FUNCTION_BLOCK FB_HE_SATT_FilterHolderTestDouble IMPLEMENTS I_HE_SATT_FilterHolder
VAR
    nNumberOfSlots : INT;
    aiFilter : ARRAY[1..PL_HE_SATT_Parameters.nMaxNumFiltersPerHolder] Of I_HE_SATT_Filter;
END_VAR


METHOD PUBLIC GetFilter : I_HE_SATT_Filter
VAR_INPUT
	nFilterNumber	: INT;
END_VAR

GetFilter := THIS^.aiFilter[nFilterNumber];
END_METHOD


PROPERTY NumberOfSlots : INT
GET

NumberOfSlots := THIS^.nNumberOfSlots;
END_GET
SET

THIS^.nNumberOfSlots := NumberOfSlots;
END_SET
END_PROPERTY


METHOD PUBLIC SetFilter
VAR_INPUT
	nFilterNumber : INT;
    iFilter : I_HE_SATT_Filter;
END_VAR

THIS^.aiFilter[nFilterNumber] := iFilter;
END_METHOD

END_FUNCTION_BLOCK

(* stored: Version 1.1.0.1
   POU FB_HE_SATT_FilterHolderTestDouble: Id {cdcd1eb9-bd8a-4335-a22e-020e71cca194}, SpecialFunc None
   Method GetFilter: Id {f3113dd3-83dc-41e8-8f98-24b65c8cff42}
   Property NumberOfSlots: Id {ef65f36b-3c7e-4172-b32f-a37ed4256cd1}
   Get Get: Id {06805441-e0e5-454c-86b1-29fec17549b7}
   Set Set: Id {5d65dd31-5c2a-4e11-acdd-05afe612d3aa}
   Method SetFilter: Id {0681b4de-c29f-4596-8a7e-f634078a4db1} *)
